(* Logix 5000 project; controller VET 1756-L62 rev 19.52; software revision 19.01; part 13 of 27 *)
(* tags used below, declared in another part *)
   _Eqp : Equipo[800];
   Batch : batch[10];
   dosificador : dosif_struct[20];
   Dosificar_MAC_01 : PHASE;
   Dosificar_MAN_01 : PHASE;
   Dosificar_MIC_01 : PHASE;
   fecha_plc : DINT;
   hora_plc : DINT;
   SetDInt : DINT[500];
   TabBin : Bins_Setup;
   Timer : TIMER[500];
   vdf : VDFS[20];
(* Dosificar_MAC_01, continued *)

ROUTINE resumen_maquinas   (* ladder *)
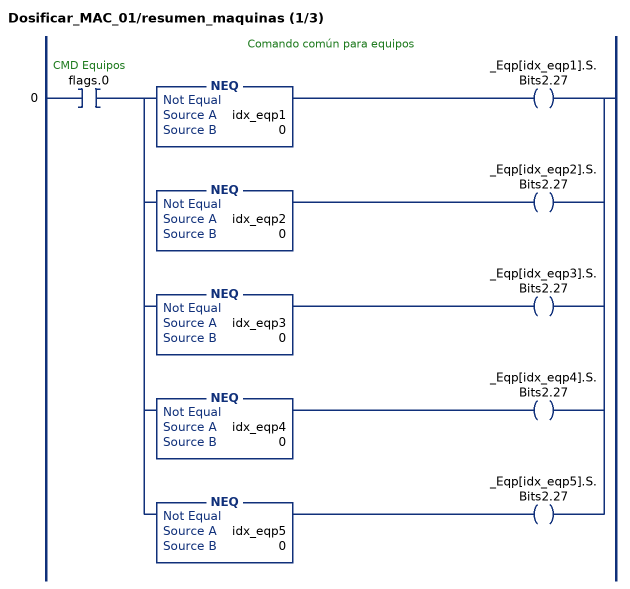
   // Comando común para equipos
   0: XIC(flags.0)[NEQ(idx_eqp1,0) OTE(_Eqp[idx_eqp1].S.Bits2.27) ,NEQ(idx_eqp2,0) OTE(_Eqp[idx_eqp2].S.Bits2.27) ,NEQ(idx_eqp3,0) OTE(_Eqp[idx_eqp3].S.Bits2.27) ,NEQ(idx_eqp4,0) OTE(_Eqp[idx_eqp4].S.Bits2.27) ,NEQ(idx_eqp5,0) OTE(_Eqp[idx_eqp5].S.Bits2.27) ];
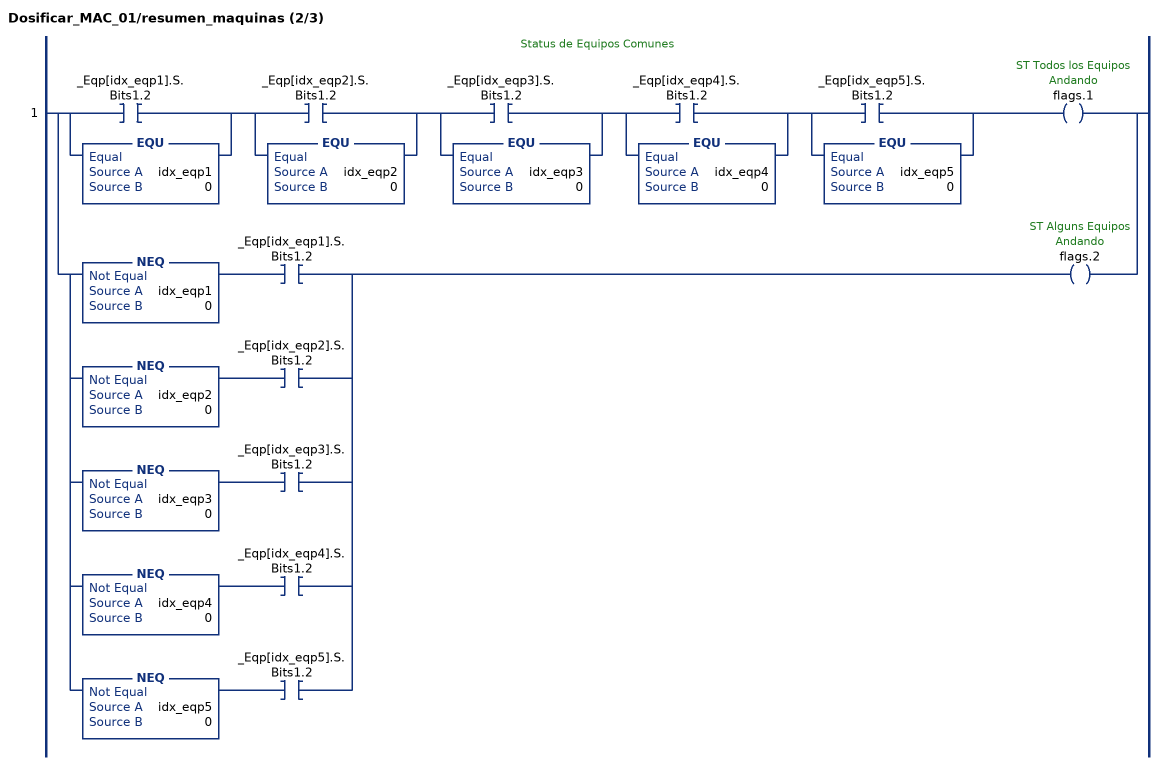
   // Status de Equipos Comunes
   1: [[XIC(_Eqp[idx_eqp1].S.Bits1.2) ,EQU(idx_eqp1,0) ] [XIC(_Eqp[idx_eqp2].S.Bits1.2) ,EQU(idx_eqp2,0) ] [XIC(_Eqp[idx_eqp3].S.Bits1.2) ,EQU(idx_eqp3,0) ] [XIC(_Eqp[idx_eqp4].S.Bits1.2) ,EQU(idx_eqp4,0) ] [XIC(_Eqp[idx_eqp5].S.Bits1.2) ,EQU(idx_eqp5,0) ] OTE(flags.1) ,[NEQ(idx_eqp1,0) XIC(_Eqp[idx_eqp1].S.Bits1.2) ,NEQ(idx_eqp2,0) XIC(_Eqp[idx_eqp2].S.Bits1.2) ,NEQ(idx_eqp3,0) XIC(_Eqp[idx_eqp3].S.Bits1.2) ,NEQ(idx_eqp4,0) XIC(_Eqp[idx_eqp4].S.Bits1.2) ,NEQ(idx_eqp5,0) XIC(_Eqp[idx_eqp5].S.Bits1.2) ] OTE(flags.2) ];
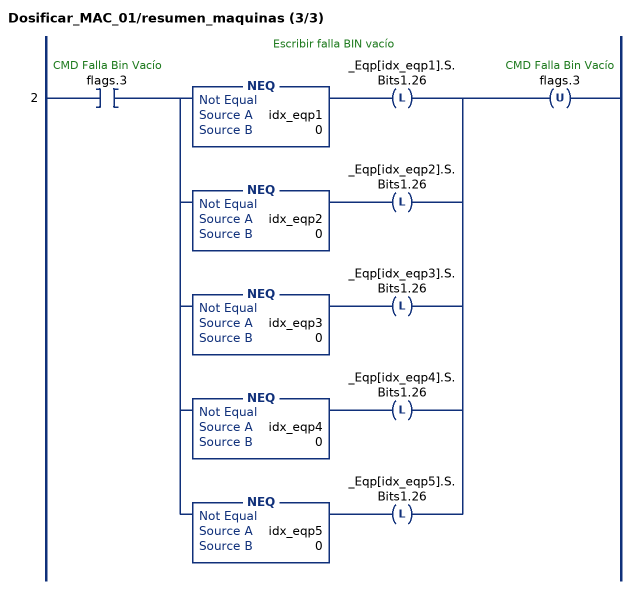
   // Escribir falla BIN vacío
   2: XIC(flags.3)[NEQ(idx_eqp1,0) OTL(_Eqp[idx_eqp1].S.Bits1.26) ,NEQ(idx_eqp2,0) OTL(_Eqp[idx_eqp2].S.Bits1.26) ,NEQ(idx_eqp3,0) OTL(_Eqp[idx_eqp3].S.Bits1.26) ,NEQ(idx_eqp4,0) OTL(_Eqp[idx_eqp4].S.Bits1.26) ,NEQ(idx_eqp5,0) OTL(_Eqp[idx_eqp5].S.Bits1.26) ]OTU(flags.3);
END_ROUTINE

ROUTINE Running   (* ladder *)
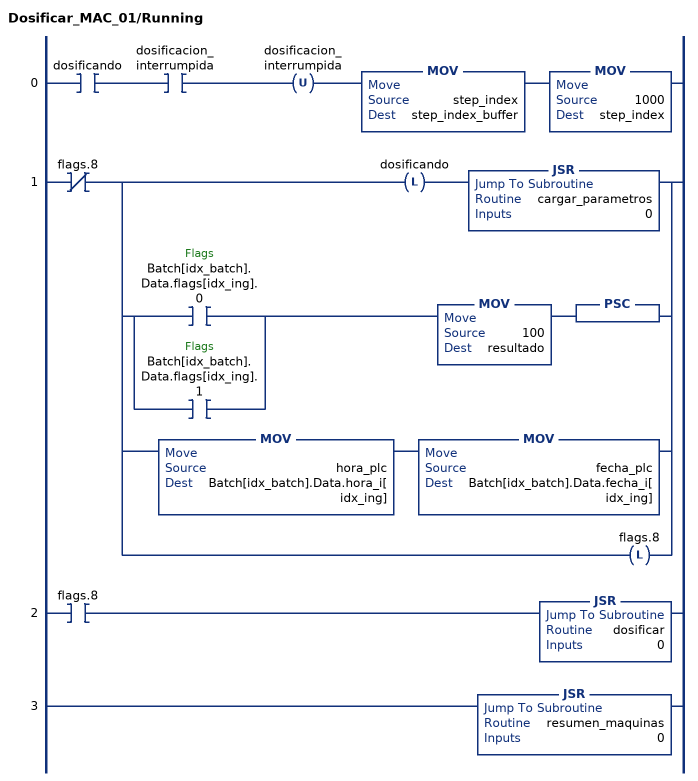
   0: XIC(dosificando)XIC(dosificacion_interrumpida)OTU(dosificacion_interrumpida)MOV(step_index,step_index_buffer)MOV(1000,step_index);
   1: XIO(flags.8)[OTL(dosificando) JSR(cargar_parametros,0) ,[[XIC(Batch[idx_batch].Data.flags[idx_ing].0) ,XIC(Batch[idx_batch].Data.flags[idx_ing].1) ] MOV(100,resultado) PSC() ,MOV(hora_plc,Batch[idx_batch].Data.hora_i[idx_ing]) MOV(fecha_plc,Batch[idx_batch].Data.fecha_i[idx_ing]) ] ,OTL(flags.8) ];
   2: XIC(flags.8)JSR(dosificar,0);
   3: JSR(resumen_maquinas,0);
END_ROUTINE
END_PROGRAM

PROGRAM Dosificar_MAN_01   (* fault routine Falla *)
VAR
   codigo_ingr : DINT;
   dosif_struct : ALIAS FOR dosificador[4];
   dosificacion_interrumpida : BOOL := 1;
   dosificando : BOOL := 1;
   error_kg : REAL;
   error_per : REAL;
   falla_struct : falla_aux;
   flags : DINT := 2;
        .0   // CMD Equipos
        .1   // ST Todos los Equipos Andando
        .2   // ST Alguns Equipos Andando
        .3   // CMD Falla Bin Vacío
        .6   // Bit Precorte
        .7   // Aplicar Precorte
   idx_batch : DINT;
   idx_bin : DINT;
   idx_ing : DINT;
   idx_tabbin : DINT := 1;
   idx_tolv : DINT;   // Índice de Tolva
   limite_err_inf : REAL := 8.0;
   limite_err_sup : REAL := 8.0;
   mensaje : ALIAS FOR dosif_struct.msg;
        .3   // Manual
        .1   // Bin Vacío
        .2   // Predescarga
        .4   // Peso Neto Negativo
        .0   // Error de Pesaje
        .5   // Dosificación interrumpida
   peso_medido : ALIAS FOR dosif_struct.peso_terreno;
   peso_neto : REAL;
   peso_objetivo : REAL := 8.0;
   respuesta : ALIAS FOR dosif_struct.ans;
        .9   // Abortar Batch
        .3   // Reintentar Misma Tolva
        .6   // Abortar Ingrediente
        .0   // Aceptar Error
        .10   // Abortar Ingrediente
        .1   // Abortar Batch
        .2   // Abortar Ingrediente
        .11   // Dosificación Completa
        .5   // Abortar Batch
        .8   // Aceptar Predescarga
        .4   // Cambiar Tolva
        .14   // Continuar Dosificación
        .16   // Abortar Ingrediente
        .7   // Pasar a Manual
        .15   // Abortar Dosificación
        .12   // Habilitar Aceptar
        .13   // Peso Neto Cero - Aceptar y Tarar
   resultado : ALIAS FOR dosif_struct.resultado;
   step_index : DINT;
   step_index_buffer : DINT;
   T : TIMER[15] := ([0].PRE := 1000, [1].PRE := 30000, [2].PRE := 3000, [3].PRE := 8000, [4].PRE := 1000, [5].PRE := 1000, [6].PRE := 1000, [7].PRE := 2500, [8].PRE := 1000, [9].PRE := 1000, [10].PRE := 5000);
   tara : REAL;
END_VAR

ROUTINE Aborting   (* ladder *)
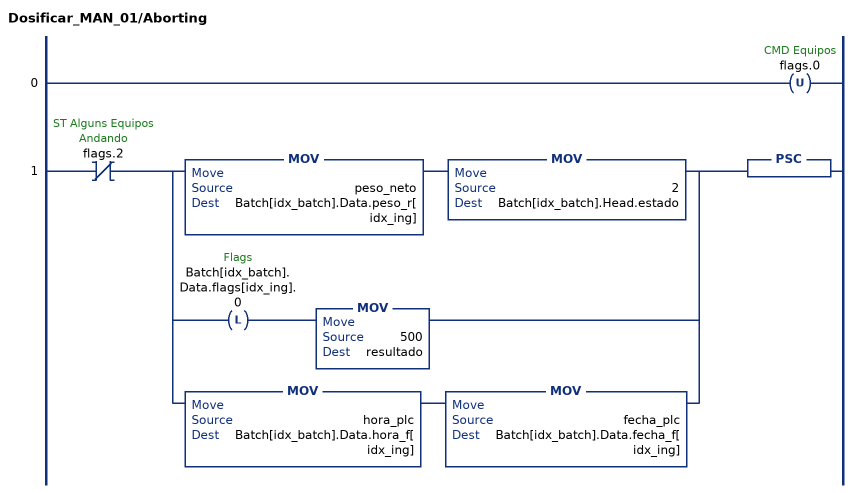
   0: OTU(flags.0);
   1: XIO(flags.2)[MOV(peso_neto,Batch[idx_batch].Data.peso_r[idx_ing]) MOV(2,Batch[idx_batch].Head.estado) ,OTL(Batch[idx_batch].Data.flags[idx_ing].0) MOV(500,resultado) ,MOV(hora_plc,Batch[idx_batch].Data.hora_f[idx_ing]) MOV(fecha_plc,Batch[idx_batch].Data.fecha_f[idx_ing]) ]PSC();
END_ROUTINE

ROUTINE cargar_parametros   (* ladder *)
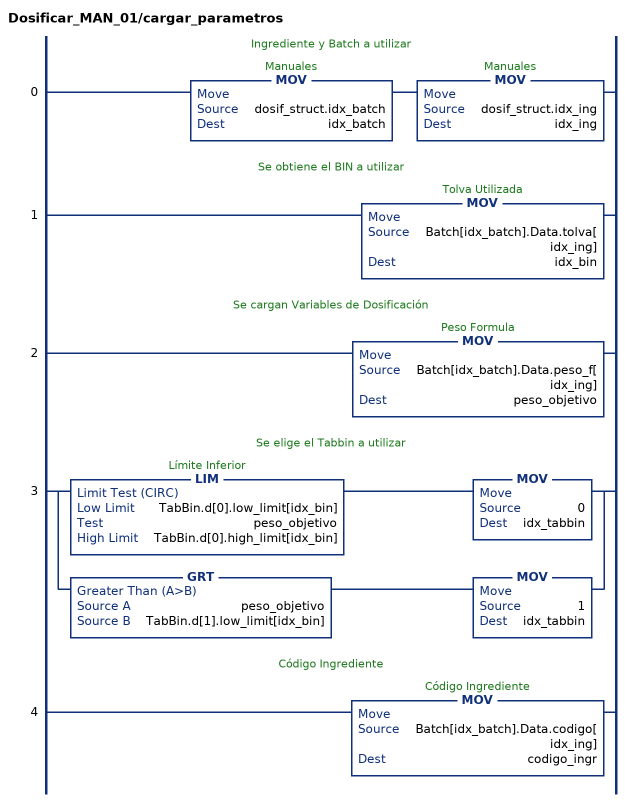
   // Ingrediente y Batch a utilizar
   0: MOV(dosif_struct.idx_batch,idx_batch)MOV(dosif_struct.idx_ing,idx_ing);
   // Se obtiene el BIN a utilizar
   1: MOV(Batch[idx_batch].Data.tolva[idx_ing],idx_bin);
   // Se cargan Variables de Dosificación
   2: MOV(Batch[idx_batch].Data.peso_f[idx_ing],peso_objetivo);
   // Se elige el Tabbin a utilizar
   3: [LIM(TabBin.d[0].low_limit[idx_bin],peso_objetivo,TabBin.d[0].high_limit[idx_bin]) MOV(0,idx_tabbin) ,GRT(peso_objetivo,TabBin.d[1].low_limit[idx_bin]) MOV(1,idx_tabbin) ];
   // Código Ingrediente
   4: MOV(Batch[idx_batch].Data.codigo[idx_ing],codigo_ingr);
END_ROUTINE

ROUTINE dosificar   (* ladder *)
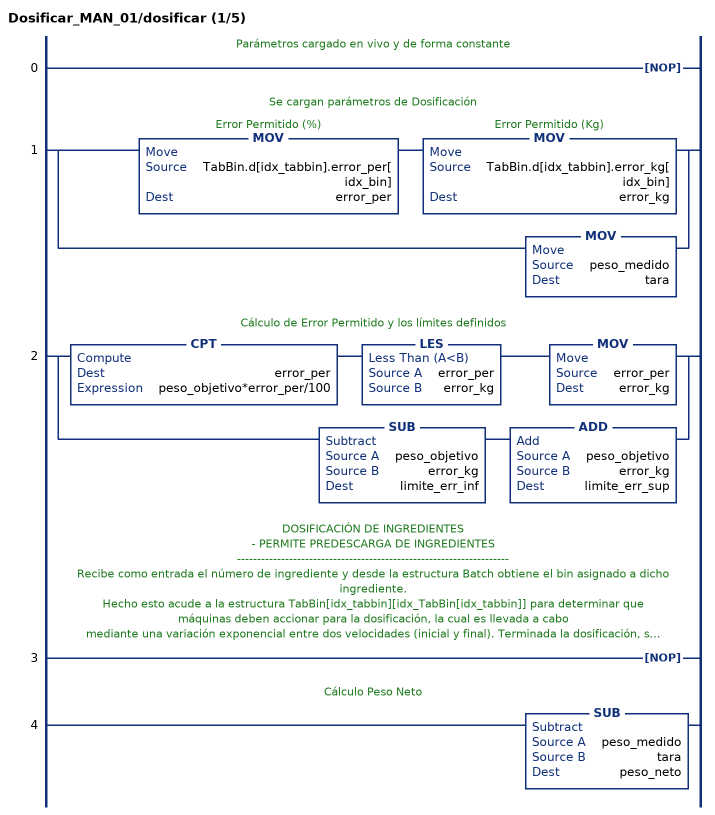
   // Parámetros cargado en vivo y de forma constante
   0: NOP();
   // Se cargan parámetros de Dosificación
   1: [MOV(TabBin.d[idx_tabbin].error_per[idx_bin],error_per) MOV(TabBin.d[idx_tabbin].error_kg[idx_bin],error_kg) ,MOV(peso_medido,tara) ];
   // Cálculo de Error Permitido y los límites definidos
   2: [CPT(error_per,peso_objetivo*error_per/100) LES(error_per,error_kg) MOV(error_per,error_kg) ,SUB(peso_objetivo,error_kg,limite_err_inf) ADD(peso_objetivo,error_kg,limite_err_sup) ];
   // DOSIFICACIÓN DE INGREDIENTES
   // - PERMITE PREDESCARGA DE INGREDIENTES
   // --------------------------------------------------------------------
   // Recibe como entrada el número de ingrediente y desde la estructura Batch obtiene el bin asignado a dicho ingrediente.
   // Hecho esto acude a la estructura TabBin[idx_tabbin][idx_TabBin[idx_tabbin]] para determinar que máquinas deben accionar para la dosificación, la cual es llevada a cabo
   // mediante una variación exponencial entre dos velocidades (inicial y final). Terminada la dosificación, se retornan o consolidan los aprendizajes
   // prBatchios de la dosificación, reflejados en un precorte ajustado.
   3: NOP();
   // Cálculo Peso Neto
   4: SUB(peso_medido,tara,peso_neto);
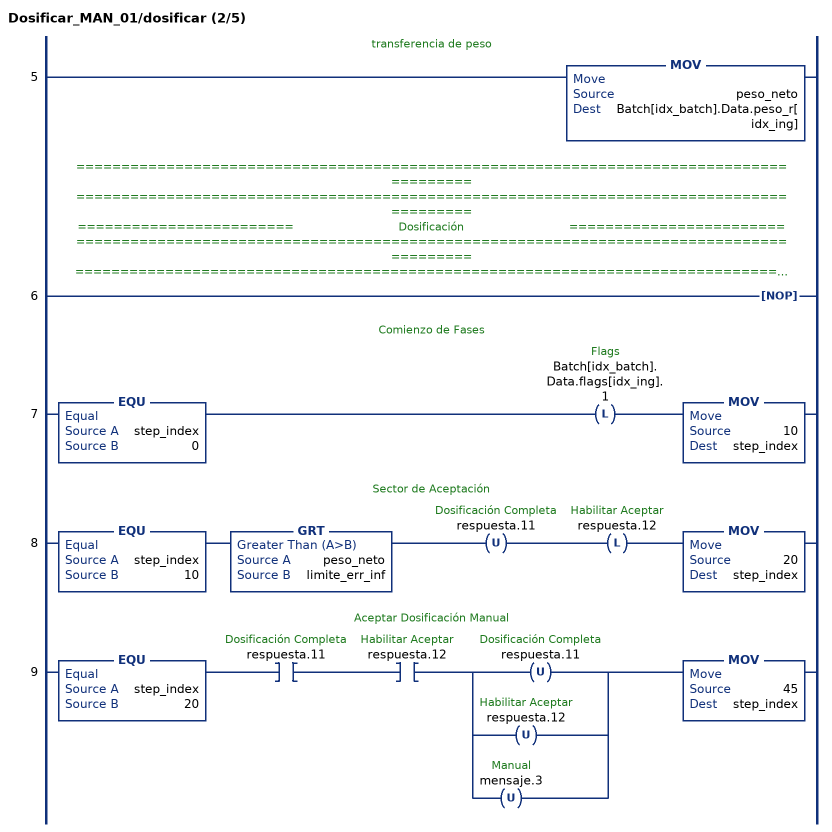
   // transferencia de peso
   5: MOV(peso_neto,Batch[idx_batch].Data.peso_r[idx_ing]);
   // ========================================================================================
   // ========================================================================================
   // ========================                              Dosificación                              ========================
   // ========================================================================================
   // ========================================================================================
   6: NOP();
   // Comienzo de Fases
   7: EQU(step_index,0)OTL(Batch[idx_batch].Data.flags[idx_ing].1)MOV(10,step_index);
   // Sector de Aceptación
   8: EQU(step_index,10)GRT(peso_neto,limite_err_inf)OTU(respuesta.11)OTL(respuesta.12)MOV(20,step_index);
   // Aceptar Dosificación Manual
   9: EQU(step_index,20)XIC(respuesta.11)XIC(respuesta.12)[OTU(respuesta.11) ,OTU(respuesta.12) ,OTU(mensaje.3) ]MOV(45,step_index);
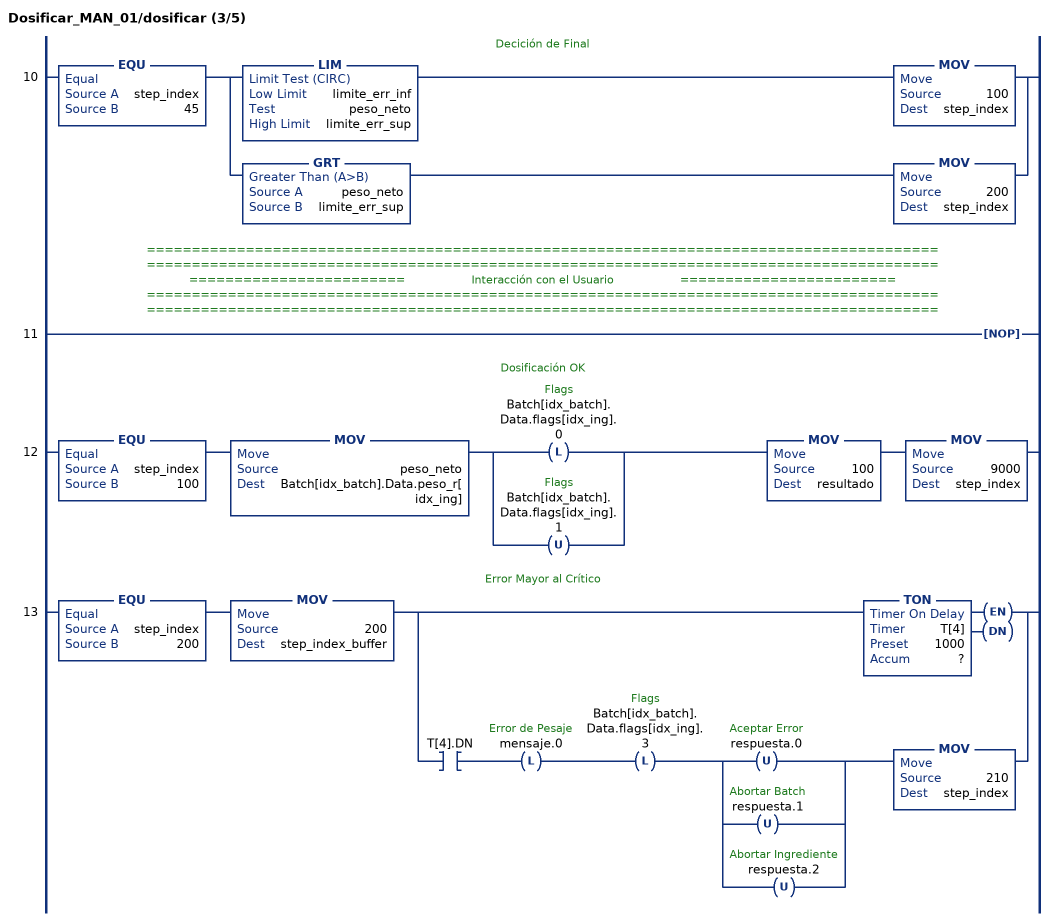
   // Decición de Final
   10: EQU(step_index,45)[LIM(limite_err_inf,peso_neto,limite_err_sup) MOV(100,step_index) ,GRT(peso_neto,limite_err_sup) MOV(200,step_index) ];
   // ========================================================================================
   // ========================================================================================
   // ========================                   Interacción con el Usuario                   ========================
   // ========================================================================================
   // ========================================================================================
   11: NOP();
   // Dosificación OK
   12: EQU(step_index,100)MOV(peso_neto,Batch[idx_batch].Data.peso_r[idx_ing])[OTL(Batch[idx_batch].Data.flags[idx_ing].0) ,OTU(Batch[idx_batch].Data.flags[idx_ing].1) ]MOV(100,resultado)MOV(9000,step_index);
   // Error Mayor al Crítico
   13: EQU(step_index,200)MOV(200,step_index_buffer)[TON(T[4],?,?) ,XIC(T[4].DN) OTL(mensaje.0) OTL(Batch[idx_batch].Data.flags[idx_ing].3) [OTU(respuesta.0) ,OTU(respuesta.1) ,OTU(respuesta.2) ] MOV(210,step_index) ];
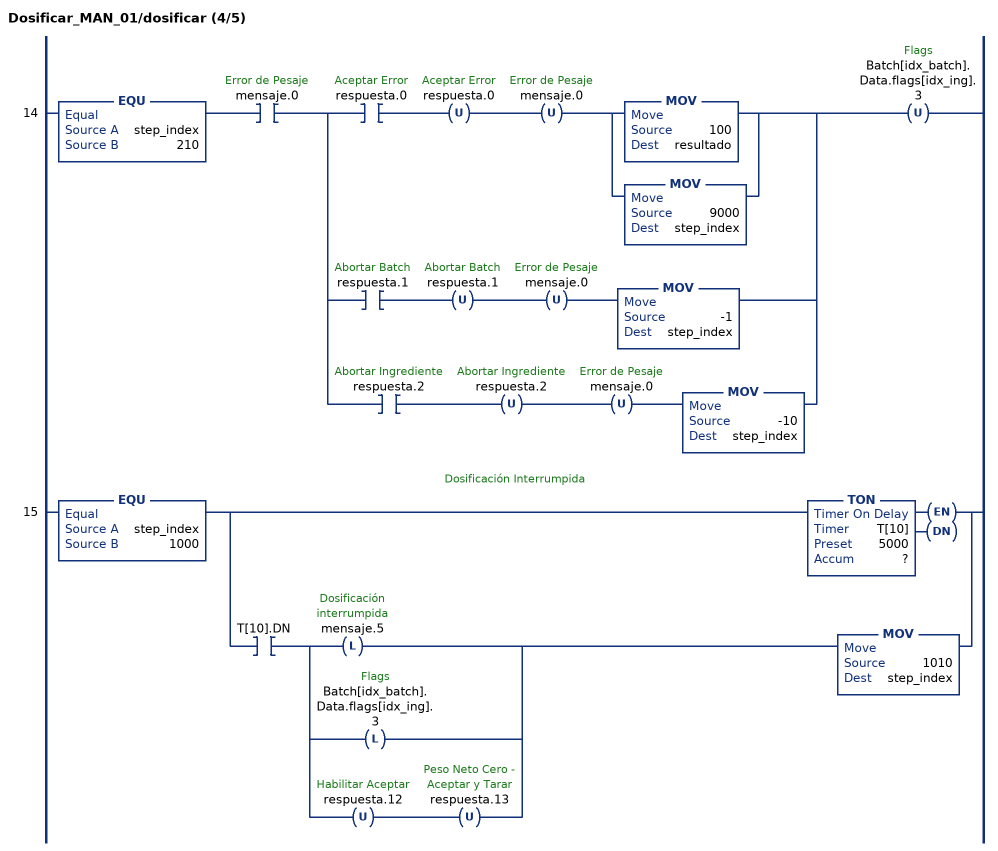
   14: EQU(step_index,210)XIC(mensaje.0)[XIC(respuesta.0) OTU(respuesta.0) OTU(mensaje.0) [MOV(100,resultado) ,MOV(9000,step_index) ] ,XIC(respuesta.1) OTU(respuesta.1) OTU(mensaje.0) MOV(-1,step_index) ,XIC(respuesta.2) OTU(respuesta.2) OTU(mensaje.0) MOV(-10,step_index) ]OTU(Batch[idx_batch].Data.flags[idx_ing].3);
   // Dosificación Interrumpida
   15: EQU(step_index,1000)[TON(T[10],?,?) ,XIC(T[10].DN) [OTL(mensaje.5) ,OTL(Batch[idx_batch].Data.flags[idx_ing].3) ,OTU(respuesta.12) OTU(respuesta.13) ] MOV(1010,step_index) ];
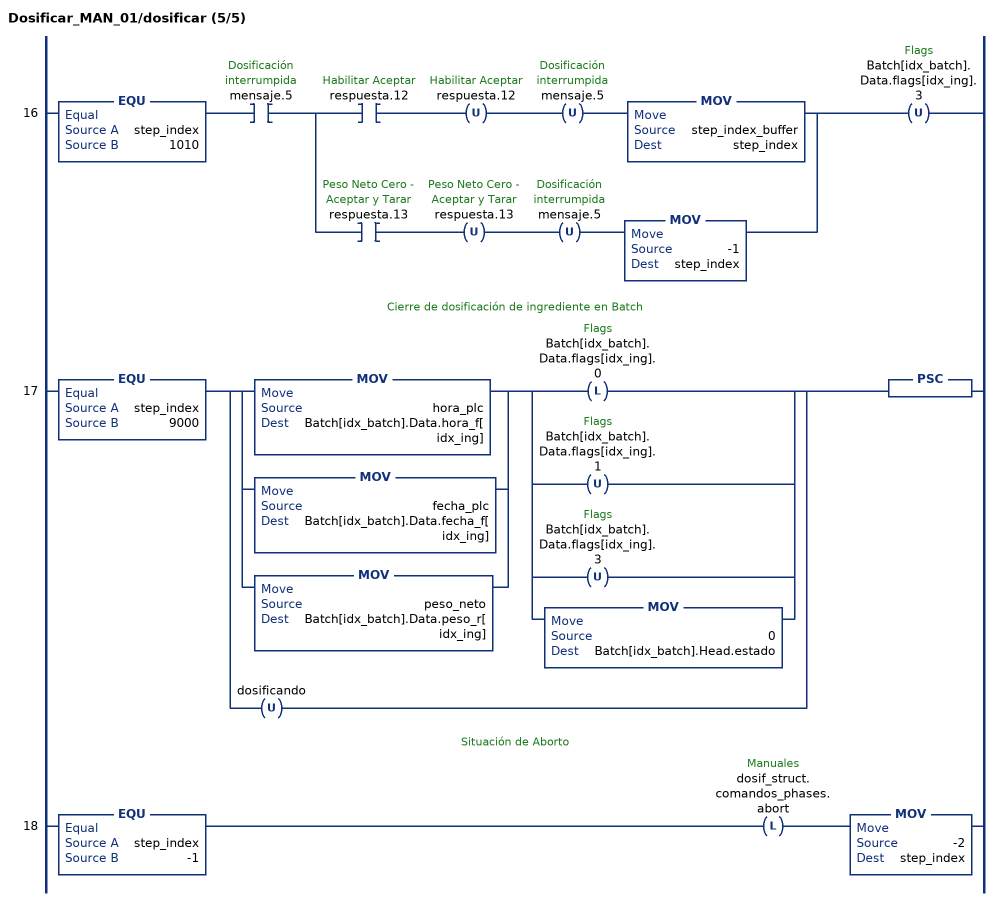
   16: EQU(step_index,1010)XIC(mensaje.5)[XIC(respuesta.12) OTU(respuesta.12) OTU(mensaje.5) MOV(step_index_buffer,step_index) ,XIC(respuesta.13) OTU(respuesta.13) OTU(mensaje.5) MOV(-1,step_index) ]OTU(Batch[idx_batch].Data.flags[idx_ing].3);
   // Cierre de dosificación de ingrediente en Batch
   17: EQU(step_index,9000)[[MOV(hora_plc,Batch[idx_batch].Data.hora_f[idx_ing]) ,MOV(fecha_plc,Batch[idx_batch].Data.fecha_f[idx_ing]) ,MOV(peso_neto,Batch[idx_batch].Data.peso_r[idx_ing]) ] [OTL(Batch[idx_batch].Data.flags[idx_ing].0) ,OTU(Batch[idx_batch].Data.flags[idx_ing].1) ,OTU(Batch[idx_batch].Data.flags[idx_ing].3) ,MOV(0,Batch[idx_batch].Head.estado) ] ,OTU(dosificando) ]PSC();
   // Situación de Aborto
   18: EQU(step_index,-1)OTL(dosif_struct.comandos_phases.abort)MOV(-2,step_index);
END_ROUTINE

ROUTINE Falla   (* ladder *)
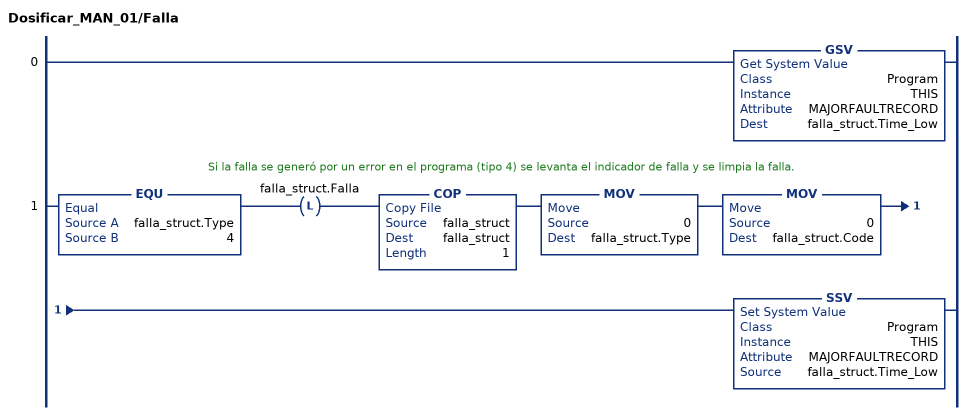
   0: GSV(Program,THIS,MAJORFAULTRECORD,falla_struct.Time_Low);
   // Si la falla se generó por un error en el programa (tipo 4) se levanta el indicador de falla y se limpia la falla.
   1: EQU(falla_struct.Type,4)OTL(falla_struct.Falla)COP(falla_struct,falla_struct,1)MOV(0,falla_struct.Type)MOV(0,falla_struct.Code)SSV(Program,THIS,MAJORFAULTRECORD,falla_struct.Time_Low);
END_ROUTINE

ROUTINE Holding   (* ladder *)
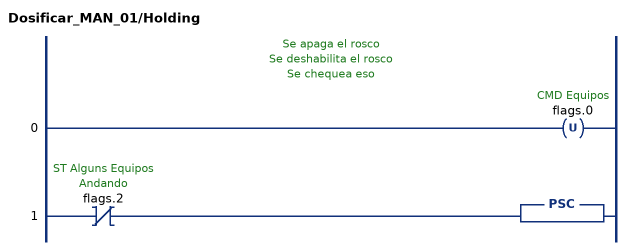
   // Se apaga el rosco
   // Se deshabilita el rosco
   // Se chequea eso
   0: OTU(flags.0);
   1: XIO(flags.2)PSC();
END_ROUTINE

ROUTINE preState   (* ladder *)
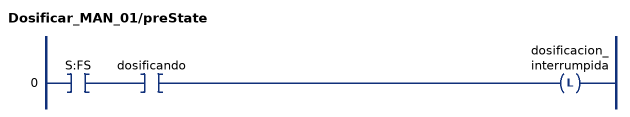
   0: XIC(S:FS)XIC(dosificando)OTL(dosificacion_interrumpida);
END_ROUTINE

ROUTINE Resetting   (* ladder *)
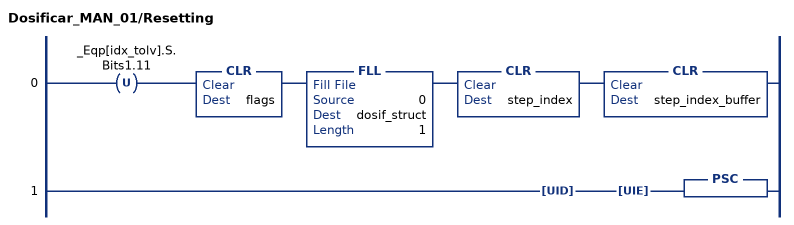
   0: OTU(_Eqp[idx_tolv].S.Bits1.11)CLR(flags)FLL(0,dosif_struct,1)CLR(step_index)CLR(step_index_buffer);
   1: UID()UIE()PSC();
END_ROUTINE

ROUTINE Restarting   (* ladder *)
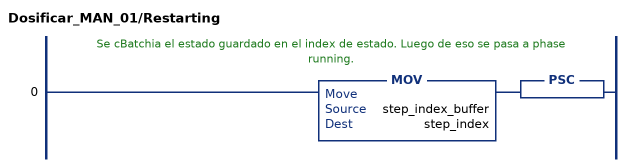
   // Se cBatchia el estado guardado en el index de estado. Luego de eso se pasa a phase running.
   0: MOV(step_index_buffer,step_index)PSC();
END_ROUTINE

ROUTINE Running   (* ladder *)
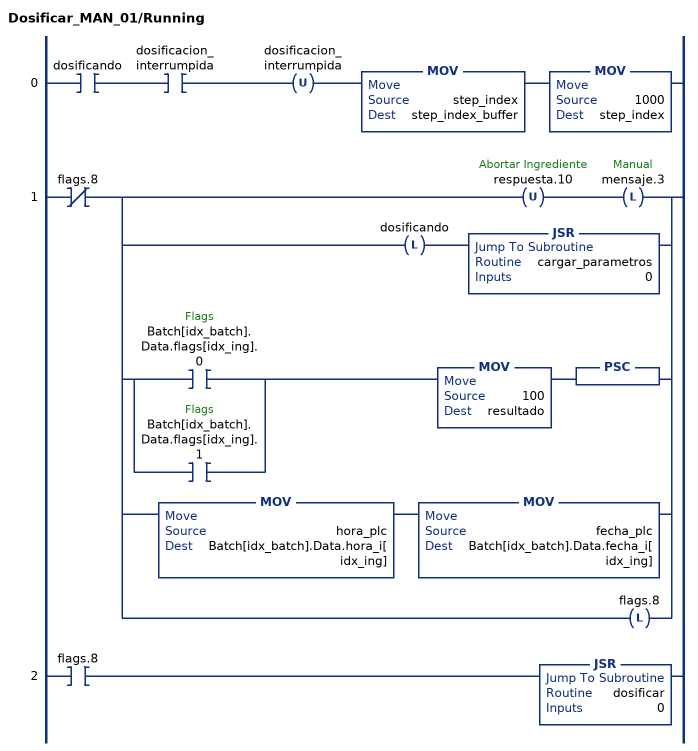
   0: XIC(dosificando)XIC(dosificacion_interrumpida)OTU(dosificacion_interrumpida)MOV(step_index,step_index_buffer)MOV(1000,step_index);
   1: XIO(flags.8)[OTU(respuesta.10) OTL(mensaje.3) ,OTL(dosificando) JSR(cargar_parametros,0) ,[[XIC(Batch[idx_batch].Data.flags[idx_ing].0) ,XIC(Batch[idx_batch].Data.flags[idx_ing].1) ] MOV(100,resultado) PSC() ,MOV(hora_plc,Batch[idx_batch].Data.hora_i[idx_ing]) MOV(fecha_plc,Batch[idx_batch].Data.fecha_i[idx_ing]) ] ,OTL(flags.8) ];
   2: XIC(flags.8)JSR(dosificar,0);
END_ROUTINE
END_PROGRAM

PROGRAM Dosificar_MIC_01   (* fault routine Falla *)
VAR
   _vel_exp : velocidad_exp := (x := 0.0034942627, curvatura := 1.0, V_inicial := 70.0, V_final := 50.0, V_salida := 50.110054);
   bufferF : REAL[5] := ([0] := 12.01828, [1] := -0.01828003, [2] := 0.0034942627);
        [2]   // Diferencia entre peso actual y objetivo
   debug : BOOL;
   dosif_extra_ingr : DINT := -1;   // Código del ingrediente que puede ser dosificado extra.
   dosif_struct : ALIAS FOR dosificador[2];
   dosificacion_interrumpida : BOOL;
   dosificando : BOOL;
   error_kg : REAL := 0.1;
   error_per : REAL := 0.6;
   falla_struct : falla_aux;
   flags : DINT;
        .1   // ST Todos los Equipos Andando
        .0   // CMD Equipos
        .2   // ST Alguns Equipos Andando
        .3   // CMD Falla Bin Vacío
        .6   // Bit Precorte
        .7   // Aplicar Precorte
   frq : ALIAS FOR dosif_struct.frq_terreno;
   frq_calculada : REAL := 50.0;
   frq_final : REAL := 50.0;
   frq_inicial : REAL := 70.0;
   hist_precorte : REAL[10] := ([0] := 1.0, [1] := 1.0, [2] := 1.0, [3] := 1.0, [4] := 1.0);
   i_fn : DINT;
   idx_batch : DINT := 3;
   idx_bin : DINT := 24;
   idx_dosif : DINT;   // Índice de dosificador usado
   idx_eqp1 : DINT := 86;
   idx_eqp2 : DINT;
   idx_eqp3 : DINT;
   idx_eqp4 : DINT;
   idx_eqp5 : DINT;
   idx_ing : DINT := 11;
   idx_tabbin : DINT := 1;
   idx_tolv : DINT := 66;   // Índice de Tolva
   limite_err_inf : REAL := 11.9;
   limite_err_sup : REAL := 12.1;
   mensaje : ALIAS FOR dosif_struct.msg;
        .3   // Manual
        .1   // Bin Vacío
        .2   // Predescarga
        .4   // Peso Neto Negativo
        .0   // Error de Pesaje
        .5   // Dosificación interrumpida
   peso_delta : REAL;
   peso_detencion : REAL := 11.958246;
   peso_intermedio : REAL := 6.0;   // Peso límite para dosificación a frecuencia máxima
   peso_max : REAL := 150.0;
   peso_medido : ALIAS FOR dosif_struct.peso_terreno;
   peso_neto : REAL := 12.01828;
   peso_neto_aux : REAL;   // Peso Neto Guardado en caso de Vaciado y llenado de tolva
   peso_objetivo : REAL := 12.0;
   precorte : REAL := 0.046323393;
   respuesta : ALIAS FOR dosif_struct.ans;
        .13   // Peso Neto Cero - Aceptar y Tarar
        .12   // Habilitar Aceptar
        .3   // Reintentar Misma Tolva
        .6   // Abortar Ingrediente
        .0   // Aceptar Error
        .10   // Abortar Ingrediente
        .9   // Abortar Batch
        .1   // Abortar Batch
        .2   // Abortar Ingrediente
        .11   // Dosificación Completa
        .5   // Abortar Batch
        .8   // Aceptar Predescarga
        .4   // Cambiar Tolva
        .14   // Continuar Dosificación
        .16   // Abortar Ingrediente
        .7   // Pasar a Manual
        .15   // Abortar Dosificación
   resultado : ALIAS FOR dosif_struct.resultado;
   return_fn : DINT;
   setD : DINT[5] := ([0] := 1, [1] := 44, [2] := 2, [3] := 1, [4] := 32);
        [1].8   // Con VDF
        [1].0   // Tipo LIW
        [4]   // Destino
        [1].2   // Predescarga
        [0]   // Mínima variación de peso para detección de tolva vacía.
        [1].3   // Aplicar Precorte
        [1].4   // Con Bloqueo de Tolva
        [1].5   // No respeta receta
        [2]   // Mezcladora izquierda
        [3]   // Mezcladora derecha
   setF : REAL[5] := ([0] := 0.1);
        [0]   // Límite para variación de peso
        [1]   // Límite para peso negativo
   step_index : DINT;
   step_index_buffer : DINT;
   T : TIMER[15] := ([0].PRE := 1000, [0].ACC := 648, [0].EN := 1, [0].TT := 1, [1].PRE := 30000, [2].PRE := 3000, [2].ACC := 3001, [2].EN := 1, [2].DN := 1, [3].PRE := 6000, [4].PRE := 1000, [5].PRE := 1000, [6].PRE := 1000, [7].PRE := 2500, [8].PRE := 1000, [9].PRE := 1000, [10].PRE := 5000);
   t_espera : DINT := 3000;
   t_pulso : DINT := 6000;
   tara : REAL := 128.60373;
END_VAR

ROUTINE _fn_dividir_ingrediente   (* ladder *)
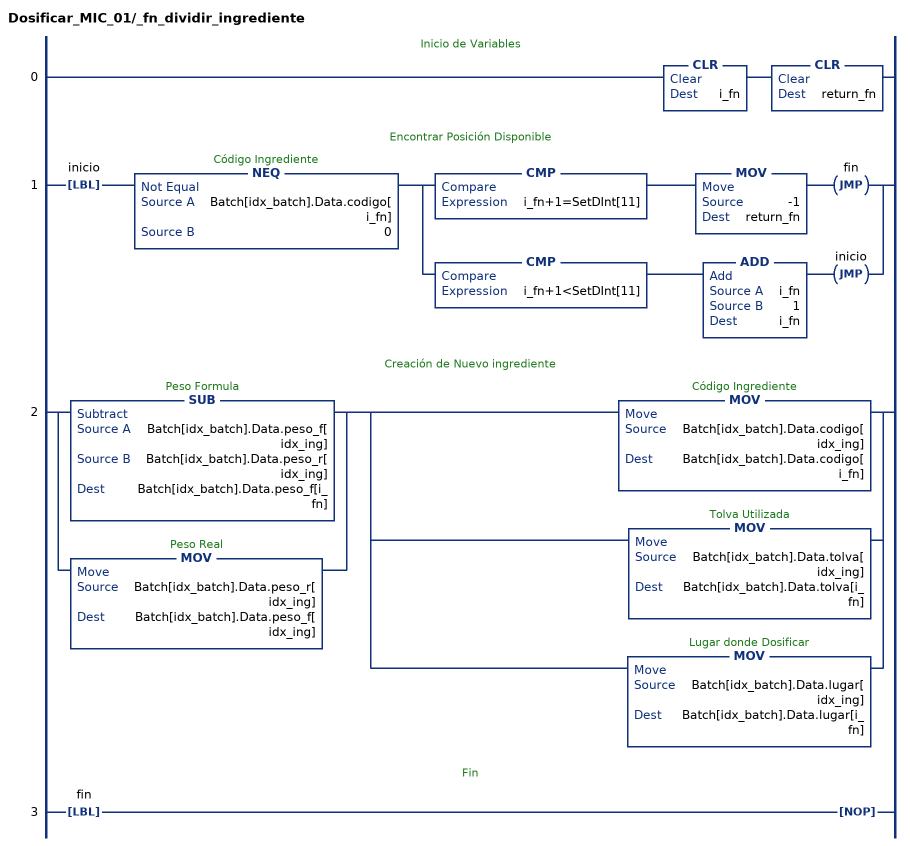
   // Inicio de Variables
   0: CLR(i_fn)CLR(return_fn);
   // Encontrar Posición Disponible
   1: LBL(inicio)NEQ(Batch[idx_batch].Data.codigo[i_fn],0)[CMP(i_fn+1=SetDInt[11]) MOV(-1,return_fn) JMP(fin) ,CMP(i_fn+1<SetDInt[11]) ADD(i_fn,1,i_fn) JMP(inicio) ];
   // Creación de Nuevo ingrediente
   2: [SUB(Batch[idx_batch].Data.peso_f[idx_ing],Batch[idx_batch].Data.peso_r[idx_ing],Batch[idx_batch].Data.peso_f[i_fn]) ,MOV(Batch[idx_batch].Data.peso_r[idx_ing],Batch[idx_batch].Data.peso_f[idx_ing]) ][MOV(Batch[idx_batch].Data.codigo[idx_ing],Batch[idx_batch].Data.codigo[i_fn]) ,MOV(Batch[idx_batch].Data.tolva[idx_ing],Batch[idx_batch].Data.tolva[i_fn]) ,MOV(Batch[idx_batch].Data.lugar[idx_ing],Batch[idx_batch].Data.lugar[i_fn]) ];
   // Fin
   3: LBL(fin)NOP();
END_ROUTINE
